// TIA Portal V15 export
// export: Created 2018-12-10T18:36:46.3784748Z, ExportSetting WithDefaults, WithReadOnly, DisplayName Totally Integrated Automation Portal, DisplayVersion V15 Update 2, DisplayName TIA Portal Openness, DisplayVersion V15 Update 2, DisplayName STEP 7 Professional, DisplayVersion V15 Update 2, DisplayName STEP 7 Safety, DisplayVersion V15, DisplayName WinCC Professional, DisplayVersion V15 Update 2, DisplayName SIMATIC Visualization Architect, DisplayVersion V15 Update 1
DATA_BLOCK "FGDB_ROBNAME@Sensopart"   // DB140
TITLE = Technology sensorpart / Technologie Sensorpart
{ S7_Optimized_Access := 'FALSE' }
AUTHOR : integra
FAMILY : SUB
VERSION : 0.1
// stored: AutoNumber true, CodeModifiedDate 2018-01-29T16:41:46.0152494Z, CompileDate 2018-02-20T10:24:46.7831888Z, CreationDate 2017-08-25T09:18:52.8131298Z, DBAccessibleFromOPCUA true, InstanceOfName iSF_TECH_ROBOT_SENSOPART, InstanceOfNumber 21, InstanceOfType FB, InterfaceModifiedDate 2018-01-24T13:32:26.306075Z, IsConsistent true, IsKnowHowProtected false, ModifiedDate 2018-01-29T16:41:46.0152494Z, ParameterModified 2017-08-16T11:39:17.0230525Z, StructureModified 2017-08-16T12:19:32.1868034Z, UDAEnableTagReadback false
"iSF_TECH_ROBOT_SENSOPART"
   // VAR_INPUT
   //    fct : Int;
   // END_VAR
   // VAR_OUTPUT
   //    qstop : Bool;
   //    busy : Bool;
   //    fault : Bool;
   // END_VAR
   // VAR_IN_OUT
   //    IfcFGExternal : "iUDT_IFC_SYS_EXTERNAL_ALARM";
   //    IfcTECH : "iUDT_IFC_ROBOT_TECH";
   //    In_PI_TECH : "iUDT_PI_ROBOT_ADRxx48_TECH";
   // END_VAR
   // VAR RETAIN
   //    F : Struct
   //       wrongID : Bool;
   //       measureError : Bool;
   //       outOfToleranze : Bool;
   //       validationError : Bool;
   //    END_STRUCT;
   //    Masks : Struct
   //       disableFault1_8 : Byte;
   //       prodRelevantFault1_8 : Byte;
   //    END_STRUCT;
   //    LastState : Struct
   //       fault1_8 : Byte;
   //       warning_1_8 : Byte;
   //    END_STRUCT;
   //    TECH_IN : Struct
   //       ID : Byte;
   //       camera1Active : Bool;
   //       camera1Ready : Bool;
   //       camera1OperationMode : Bool;
   //       camera1TriggerMode : Bool;
   //       camera1CalibMastered : Bool;
   //       camera2Active : Bool;
   //       camera2Ready : Bool;
   //       camera2OperationMode : Bool;
   //       camera2TriggerMode : Bool;
   //       camera2CalibMastered : Bool;
   //       measureError : Bool;
   //       outOfToleranze : Bool;
   //       validationError : Bool;
   //       qstopp : Bool;
   //       busy : Bool;
   //       technoBit16 : Bool;
   //       technoBit17 : Bool;
   //       technoBit18 : Bool;
   //       technoBit19 : Bool;
   //       technoBit20 : Bool;
   //       technoBit21 : Bool;
   //       technoBit22 : Bool;
   //       technoBit23 : Bool;
   //       technoBit24 : Bool;
   //       technoBit25 : Bool;
   //       technoBit26 : Bool;
   //       technoBit27 : Bool;
   //       technoBit28 : Bool;
   //       technoBit29 : Bool;
   //       technoBit30 : Bool;
   //       technoBit31 : Bool;
   //       technoBit32 : Bool;
   //       technoBit33 : Bool;
   //       technoBit34 : Bool;
   //       technoBit35 : Bool;
   //       technoBit36 : Bool;
   //       technoBit37 : Bool;
   //       technoBit38 : Bool;
   //       technoBit39 : Bool;
   //       technoBit40 : Bool;
   //    END_STRUCT;
   // END_VAR
BEGIN
END_DATA_BLOCK
